// TwinCAT 3 PLC project P_Connect
// ProgramVersion: 3.1.4023.0
// libraries:
//   Tc2_EIB, * (Beckhoff Automation GmbH)
//   Tc2_IoFunctions, * (Beckhoff Automation GmbH)
//   Tc2_MBus, * (Beckhoff Automation GmbH)
//   Tc2_SerialCom, * (Beckhoff Automation GmbH)
//   Tc2_Standard, * (Beckhoff Automation GmbH)
//   Tc2_System, * (Beckhoff Automation GmbH)
//   Tc3_Module, * (Beckhoff Automation GmbH)
// project tree:
//   DUTs/ st_P_Connect_to_Lynus.TcDUT
//   GVLs/ Global_var.TcGVL, GVL_EfficientIO.TcGVL, p_Datenschnittstelle.TcPOU
//   / PlcTask.TcTTO
//   POUs/ MAIN.TcPOU
// real-time tasks:
//   TASK PlcTask: cycle T#10ms, priority 20, ADS port 350
//   TASK EfficientIO_Communication: cycle T#5ms, priority 15, ADS port 351
//   TASK PlcTask1: cycle T#10ms, priority 21, ADS port 353
// variable links:
//   Lynus_Test/Lynus_Test Instance <-> P_Connect/P_Connect Instance
//     PlcTask1 Inputs/GVL.lynus_in <-> PlcTask Outputs/GVL_EfficientIO.lynus_out
//     PlcTask1 Outputs/GVL.lynus_out <-> PlcTask Inputs/GVL_EfficientIO.lynus_in

CONFIGURATION P_Connect
    RESOURCE PLC ON TwinCAT3
        TASK PlcTask(INTERVAL := T#10ms, PRIORITY := 20);
        PROGRAM MAIN WITH PlcTask : MAIN;
    END_RESOURCE
END_CONFIGURATION

// ---- DUTs/st_P_Connect_to_Lynus.TcDUT
TYPE st_P_Connect_to_Lynus :
STRUCT
	Wert_1	:REAL;	
	Wert_2	:REAL;	
	Wert_3	:REAL;	
	Wert_4	:REAL;	
	Wert_5	:REAL;	
	Wert_6	:REAL;	
	Wert_7	:BOOL;	
	Wert_8	:REAL;	
	Wert_9	:REAL;	
	Wert_10	:REAL;
	Wert_11	:REAL;	
	Wert_12	:REAL;	
	Wert_13	:REAL;	
	Wert_14	:REAL;	
	Wert_15	:REAL;	
	Wert_16	:REAL;	
	Wert_17	:REAL;	
	Wert_18	:REAL;	
	Wert_19	:REAL;	
	Wert_20	:REAL;
	Wert_21	:REAL;	
	Wert_22	:REAL;	
	Wert_23	:REAL;	
	Wert_24	:REAL;	
	Wert_25	:REAL;	
	Wert_26	:REAL;	
	Wert_27	:REAL;	
	Wert_28	:REAL;	
	Wert_29	:REAL;	
	Wert_30	:REAL;
	Wert_31	:REAL;
	Wert_32	:REAL;
	Wert_33	:REAL;
	Wert_34	:REAL;
	Wert_35	:REAL;
	Wert_36	:REAL;
	Wert_37	:REAL;
	Wert_38	:REAL;
	Wert_39	:REAL;
	Wert_40	:REAL;
	Wert_41	:BOOL;
	Wert_42	:BOOL;
	Wert_43	:BOOL;
	Wert_44	:BOOL;
	Wert_45	:BOOL;
	Wert_46	:BOOL;
	Wert_47	:BOOL;
	Wert_48	:BOOL;
	Wert_49	:BOOL;
	Wert_50	:BOOL;
	Wert_51	:BOOL;
	Wert_52	:BOOL;
END_STRUCT
END_TYPE

// ---- GVLs/Global_var.TcGVL
VAR_GLOBAL
	_ARRAY_IP			:ARRAY [1..50] OF STRING; 
	_ARRAY_name_of_var	:ARRAY [1..50] OF STRING(255);
	_ARRAY_var_value	:ARRAY [1..50] OF REAL;
END_VAR

// ---- GVLs/GVL_EfficientIO.TcGVL
{attribute 'qualified_only'}
VAR_GLOBAL
	lynus_out   				AT %Q* 	: st_P_Connect_to_Lynus;
	lynus_in   					AT %I* 	: st_P_Connect_to_Lynus;	
	
	(*KNX*)
	TEMP_INNEN_1			:REAL;	
	RH_INNEN_1				:REAL;	
	TEMP_INNEN_2			:REAL;	
	RH_INNEN_2				:REAL;	
	TEMP_AUSSEN				:REAL;	
	RH_AUSSEN				:REAL;		
	AKTIVITAET				:BOOL;
	
	(*M-Bus variablen für Lynus*)
	ELEKTRO_1_Zaehler		:REAL;
	ELEKTRO_1_Leistung		:REAL;
	ELEKTRO_2_Zaehler		:REAL;
	ELEKTRO_2_Leistung		:REAL;
	ELEKTRO_3_Zaehler		:REAL;
	ELEKTRO_3_Leistung		:REAL;
	ELEKTRO_4_Zaehler		:REAL;
	ELEKTRO_4_Leistung		:REAL;
	ELEKTRO_5_Zaehler		:REAL;
	ELEKTRO_5_Leistung		:REAL;
	HEIZEN					:REAL;
	
	(*IMPULSZÄHLER*)
	Wasseruhr_1				:REAL;
	Wasseruhr_2				:REAL;

	(*PT1000 Temp.*)
	TEMP_HKLS_1				:REAL;
	TEMP_HKLS_2				:REAL;
	TEMP_HKLS_3				:REAL;
	TEMP_HKLS_4				:REAL;
	TEMP_HKLS_5				:REAL; 
	TEMP_HKLS_6				:REAL;
	TEMP_HKLS_7				:REAL;
	TEMP_HKLS_8				:REAL;
	
	(*Zentalfunktionen*)
	VERSCHATTUNG_auf		:BOOL;
	VERSCHATTUNG_ab			:BOOL;
	ZENTRAL_LICHT_ein_EG	:BOOL;
	ZENTRAL_LICHT_aus_EG	:BOOL;
	ZENTRAL_LICHT_ein_OG	:BOOL;
	ZENTRAL_LICHT_aus_OG	:BOOL;
	BA3_ZENTRAL_LICHT_ein	:BOOL;
	BA3_ZENTRAL_LICHT_aus	:BOOL;
	BA3_VERSCHATTUNG_auf_EG	:BOOL;
	BA3_VERSCHATTUNG_ab_EG	:BOOL;
	BA3_VERSCHATTUNG_auf_OG	:BOOL;
	BA3_VERSCHATTUNG_ab_OG	:BOOL;
END_VAR

// ---- POUs/MAIN.TcPOU
PROGRAM MAIN
VAR

l_ton_Trigger_Auslesen			: TON;
l_ton_Trigger_Auslesen_BOOL		: TON;

l_tp_VERSCHATTUNG_auf		: TP;
l_tp_VERSCHATTUNG_ab		: TP;
l_tp_ZENTRAL_LICHT_ein_EG	: TP;
l_tp_ZENTRAL_LICHT_aus_EG	: TP;
l_tp_ZENTRAL_LICHT_ein_OG	: TP;
l_tp_ZENTRAL_LICHT_aus_OG	: TP;

l_BA3_tp_VERSCHATTUNG_auf_OG	: TP;
l_BA3_tp_VERSCHATTUNG_ab_OG		: TP;
l_BA3_tp_VERSCHATTUNG_auf_EG	: TP;
l_BA3_tp_VERSCHATTUNG_ab_EG		: TP;
l_BA3_tp_ZENTRAL_LICHT_ein		: TP;
l_BA3_tp_ZENTRAL_LICHT_aus		: TP;



l_fb_ADS_read_HK_LA 		: ADSRDWRTEX; 
l_fb_ADS_read_HK_LA_BOOL	: ADSRDWRTEX; 

i :INT:= 1;
l_b_only_once	:BOOL;
l_b_test		:BOOL;
l_r_destaddr	:REAL;
gv_PCon_bAktivitaet_EG_OG :BOOL;
END_VAR

_ARRAY_IP[1] := '10.0.0.10.1.1';
_ARRAY_name_of_var[1] := '.p_machineParameter_i1.ToZpoint.ProductDataAttributes_EZ_Gesamtzaehler_i1.EZ_Gesamtzaehler_Zaehlerwerte_1_ov_r_Wirkenergie_positivTotal.r_value';

_ARRAY_IP[2] := '10.0.0.10.1.1';
_ARRAY_name_of_var[2] := '.p_machineParameter_i1.ToZpoint.ProductDataAttributes_EZ_Gesamtzaehler_i1.EZ_Gesamtzaehler_Zaehlerwerte_1_ov_r_Wirkleistung_positivTotal.r_value';

_ARRAY_IP[3] := '10.0.0.10.1.1';
_ARRAY_name_of_var[3] := '.p_machineParameter_i1.ToZpoint.ProductDataAttributes_EZ_Waermepumpe_1_i1.EZ_Waermepumpe_1_Zaehlerwerte_ov_r_EnergyTotal.r_value';

_ARRAY_IP[4] := '10.0.0.10.1.1';
_ARRAY_name_of_var[4] := '.p_machineParameter_i1.ToZpoint.ProductDataAttributes_EZ_Waermepumpe_1_i1.EZ_Waermepumpe_1_Zaehlerwerte_ov_r_Wirkleistung.r_value';

_ARRAY_IP[5] := '10.0.0.10.1.1';
_ARRAY_name_of_var[5] := '.p_machineParameter_i1.ToZpoint.ProductDataAttributes_EZ_Waermepumpe_2_i1.EZ_Waermepumpe_2_Zaehlerwerte_ov_r_EnergyTotal.r_value';

_ARRAY_IP[6] := '10.0.0.10.1.1';
_ARRAY_name_of_var[6] := '.p_machineParameter_i1.ToZpoint.ProductDataAttributes_EZ_Waermepumpe_2_i1.EZ_Waermepumpe_2_Zaehlerwerte_ov_r_Wirkleistung.r_value';

_ARRAY_IP[7] := '10.0.0.10.1.1';
_ARRAY_name_of_var[7] := '.p_machineParameter_i1.ToZpoint.ProductDataAttributes_EZ_Ladestation_1_i1.EZ_Ladestation_1_Zaehlerwerte_ov_r_EnergyTotal.r_value';

_ARRAY_IP[8] := '10.0.0.10.1.1';
_ARRAY_name_of_var[8] := '.p_machineParameter_i1.ToZpoint.ProductDataAttributes_EZ_Ladestation_1_i1.EZ_Ladestation_1_Zaehlerwerte_ov_r_Wirkleistung.r_value';

_ARRAY_IP[9] := '10.0.0.10.1.1';
_ARRAY_name_of_var[9] := '.p_machineParameter_i1.ToZpoint.ProductDataAttributes_EZ_Ladestation_2_i1.EZ_Ladestation_2_Zaehlerwerte_ov_r_EnergyTotal.r_value';

_ARRAY_IP[10] := '10.0.0.10.1.1';
_ARRAY_name_of_var[10] := '.p_machineParameter_i1.ToZpoint.ProductDataAttributes_EZ_Ladestation_2_i1.EZ_Ladestation_2_Zaehlerwerte_ov_r_Wirkleistung.r_value';

_ARRAY_IP[11] := '10.0.0.10.1.1';
_ARRAY_name_of_var[11] := '.p_machineParameter_i1.ToZpoint.ProductDataAttributes_EZ_Ladestation_5_i1.EZ_Ladestation_5_Zaehlerwerte_ov_r_EnergyTotal.r_value';

_ARRAY_IP[12] := '10.0.0.10.1.1';
_ARRAY_name_of_var[12] := '.p_machineParameter_i1.ToZpoint.ProductDataAttributes_EZ_Ladestation_5_i1.EZ_Ladestation_5_Zaehlerwerte_ov_r_Wirkleistung.r_value';

_ARRAY_IP[13] := '10.0.0.10.1.1';
_ARRAY_name_of_var[13] := '.p_machineParameter_i1.ToZpoint.ProductDataAttributes_EZ_PV_Anlage_i1.EZ_PV_Wechselrichter_1_ov_r_ErzeugteWirkenergie.r_value';

_ARRAY_IP[14] := '10.0.0.10.1.1';
_ARRAY_name_of_var[14] := '.p_machineParameter_i1.ToZpoint.ProductDataAttributes_EZ_PV_Anlage_i1.EZ_PV_Wechselrichter_1_ov_r_Wirkleistung.r_value';

_ARRAY_IP[15] := '10.0.0.10.1.1';
_ARRAY_name_of_var[15] := '.p_machineParameter_i1.ToZpoint.ProductDataAttributes_EZ_PV_Anlage_i1.EZ_PV_Wechselrichter_2_ov_r_ErzeugteWirkenergie.r_value';

_ARRAY_IP[16] := '10.0.0.10.1.1';
_ARRAY_name_of_var[16] := '.p_machineParameter_i1.ToZpoint.ProductDataAttributes_EZ_PV_Anlage_i1.EZ_PV_Wechselrichter_2_ov_r_Wirkleistung.r_value';

_ARRAY_IP[17] := '10.0.0.10.1.1';
_ARRAY_name_of_var[17] := '.p_machineParameter_i1.ToZpoint.ProductDataAttributes_WMZ_01_Gaskessel_i1.WMZ_01_Gaskessel_Normaltarif_ov_r_EnergyTarif.r_value';

_ARRAY_IP[18] := '10.0.0.10.1.1';
_ARRAY_name_of_var[18] := '.p_machineParameter_i1.ToZpoint.ProductDataAttributes_WMZ_01_Gaskessel_i1.WMZ_01_Gaskessel_ov_r_Power.r_value';

_ARRAY_IP[19] := '10.0.0.10.1.1';
_ARRAY_name_of_var[19] := '.p_machineParameter_i1.ToZpoint.ProductDataAttributes_WMZ_03_WT01_WP_i1.WMZ_03_Waermetauscher_1_WP_ov_r_Power.r_value';

_ARRAY_IP[20] := '10.0.0.10.1.1';
_ARRAY_name_of_var[20] := '.p_machineParameter_i1.ToZpoint.ProductDataAttributes_WMZ_03_WT01_WP_i1.WMZ_03_Waermetauscher_1_WP_Normaltarif_ov_r_EnergyTarif.r_value';

_ARRAY_IP[21] := '10.0.0.10.1.1';
_ARRAY_name_of_var[21] := '.p_machineParameter_i1.ToZpoint.ProductDataAttributes_WMZ_03_WT01_WP_i1.WMZ_03_Waermetauscher_1_WP_Tarif_1_ov_r_EnergyTarif.r_value';

//notdonecontrolle
_ARRAY_IP[22] := '10.0.0.20.1.1';
_ARRAY_name_of_var[22] := '.p_machineParameter_i1.ToZpoint.Visualisierung_Wettersation_i1.Wettersation.Wetterstation_1.Temperatur.ov_r_Data';

_ARRAY_IP[23] := '10.0.0.20.1.1';
_ARRAY_name_of_var[23] := '.p_machineParameter_i1.ToZpoint.ProductDataAttributes_LA_Temperatursensoren_i1.LA_Temperatursensoren_Temperatur_Zuluft_ov_r_valueCorrected.r_value';

_ARRAY_IP[24] := '10.0.0.20.1.1';
_ARRAY_name_of_var[24] := '.p_machineParameter_i1.ToZpoint.ProductDataAttributes_Raum_104_Buero_2_i1.Raum_104_Buero_2_ov_rRaumtemperatur.r_value';

_ARRAY_IP[25] := '10.0.0.20.1.1';
_ARRAY_name_of_var[25] := '.p_machineParameter_i1.ToZpoint.ProductDataAttributes_Halle_027_Montage_i1.Halle_027_Montage_ov_rRaumtemperatur.r_value';

_ARRAY_IP[26] := '10.0.0.20.1.1';
_ARRAY_name_of_var[26] := '.p_machineParameter_i1.ToZpoint.ProductDataAttributes_Raum_025_Mehrzweck_und_Aufenthaltsraum_i1.Raum_025_Mehrzweck_und_Aufenthaltsraum_ov_rRaumtemperatur.r_value';

_ARRAY_IP[27] := '10.0.0.10.1.1';
_ARRAY_name_of_var[27] := '.p_machineParameter_i1.ToZpoint.ProductDataAttributes_EZ_Gesamtzaehler_i1.EZ_Gesamtzaehler_Zaehlerwerte_1_ov_r_Wirkenergie_nagativTotal.r_value';

_ARRAY_IP[28] := '10.0.0.10.1.1';
_ARRAY_name_of_var[28] := '.p_machineParameter_i1.ToZpoint.ProductDataAttributes_EZ_Gesamtzaehler_i1.EZ_Gesamtzaehler_Zaehlerwerte_1_ov_r_Wirkleistung_nagativTotal.r_value';

_ARRAY_IP[29] := '10.0.0.10.1.1';
_ARRAY_name_of_var[29] := '.p_machineParameter_i1.ToZpoint.ProductDataAttributes_EZ_PV_Anlage_i1.EZ_PV_Wechselrichter_3_ov_r_ErzeugteWirkenergie.r_value';

_ARRAY_IP[30] := '10.0.0.10.1.1';
_ARRAY_name_of_var[30] := '.p_machineParameter_i1.ToZpoint.ProductDataAttributes_EZ_PV_Anlage_i1.EZ_PV_Wechselrichter_3_ov_r_Wirkleistung.r_value';

_ARRAY_IP[31] := '10.0.0.10.1.1';
_ARRAY_name_of_var[31] := '.p_machineParameter_i1.ToZpoint.ProductDataAttributes_EZ_PV_Anlage_i1.EZ_PV_Wechselrichter_4_ov_r_ErzeugteWirkenergie.r_value';

_ARRAY_IP[32] := '10.0.0.10.1.1';
_ARRAY_name_of_var[32] := '.p_machineParameter_i1.ToZpoint.ProductDataAttributes_EZ_PV_Anlage_i1.EZ_PV_Wechselrichter_4_ov_r_Wirkleistung.r_value';

_ARRAY_IP[33] := '10.0.0.10.1.1';
_ARRAY_name_of_var[33] := '.p_machineParameter_i1.ToZpoint.ProductDataAttributes_EZ_PV_Anlage_i1.EZ_PV_Wechselrichter_5_ov_r_ErzeugteWirkenergie.r_value';

_ARRAY_IP[34] := '10.0.0.10.1.1';
_ARRAY_name_of_var[34] := '.p_machineParameter_i1.ToZpoint.ProductDataAttributes_EZ_PV_Anlage_i1.EZ_PV_Wechselrichter_5_ov_r_Wirkleistung.r_value';

_ARRAY_IP[35] := '10.0.0.10.1.1';
_ARRAY_name_of_var[35] := '.p_machineParameter_i1.ToZpoint.ProductDataAttributes_EZ_PV_Anlage_i1.EZ_PV_Wechselrichter_6_ov_r_ErzeugteWirkenergie.r_value';

_ARRAY_IP[36] := '10.0.0.10.1.1';
_ARRAY_name_of_var[36] := '.p_machineParameter_i1.ToZpoint.ProductDataAttributes_EZ_PV_Anlage_i1.EZ_PV_Wechselrichter_6_ov_r_Wirkleistung.r_value';

_ARRAY_IP[37] := '10.0.0.10.1.1';
_ARRAY_name_of_var[37] := '.p_machineParameter_i1.ToZpoint.ProductDataAttributes_EZ_PV_Anlage_i1.EZ_PV_Wechselrichter_7_ov_r_ErzeugteWirkenergie.r_value';

_ARRAY_IP[38] := '10.0.0.10.1.1';
_ARRAY_name_of_var[38] := '.p_machineParameter_i1.ToZpoint.ProductDataAttributes_EZ_PV_Anlage_i1.EZ_PV_Wechselrichter_7_ov_r_Wirkleistung.r_value';

_ARRAY_IP[39] := '10.0.0.10.1.1';
_ARRAY_name_of_var[39] := '.p_machineParameter_i1.ToZpoint.ProductDataAttributes_EZ_PV_Anlage_i1.EZ_PV_Wechselrichter_8_ov_r_ErzeugteWirkenergie.r_value';

_ARRAY_IP[40] := '10.0.0.10.1.1';
_ARRAY_name_of_var[40] := '.p_machineParameter_i1.ToZpoint.ProductDataAttributes_EZ_PV_Anlage_i1.EZ_PV_Wechselrichter_8_ov_r_Wirkleistung.r_value';

_ARRAY_IP[41] := '10.0.0.10.1.1';
_ARRAY_name_of_var[41] := '.p_machineParameter_i1.ToZpoint.ProductDataAttributes_EZ_PV_Anlage_i1.EZ_PV_Wechselrichter_9_ov_r_ErzeugteWirkenergie.r_value';

_ARRAY_IP[42] := '10.0.0.10.1.1';
_ARRAY_name_of_var[42] := '.p_machineParameter_i1.ToZpoint.ProductDataAttributes_EZ_PV_Anlage_i1.EZ_PV_Wechselrichter_9_ov_r_Wirkleistung.r_value';

//BA3 WP aktulle leistung
_ARRAY_IP[43] := '10.0.0.30.1.1';
_ARRAY_name_of_var[43] := '.p_machineParameter_i1.ToZpoint.ProductDataAttributes_WMZ02_Waermepumpe_BA3E_i1.WMZ02_Waermepumpe_BA3E_ov_r_Power.r_value'; 
//BA3 WP Wärme Energie
_ARRAY_IP[44] := '10.0.0.30.1.1';
_ARRAY_name_of_var[44] := '.p_machineParameter_i1.ToZpoint.ProductDataAttributes_WMZ02_Waermepumpe_BA3E_i1.WMZ02_Waermepumpe_BA3E_ov_r_EnergyT1.r_value';
//BA3 Kälte Energie
_ARRAY_IP[45] := '10.0.0.30.1.1';
_ARRAY_name_of_var[45] := '.p_machineParameter_i1.ToZpoint.ProductDataAttributes_WMZ02_Waermepumpe_BA3E_i1.WMZ02_Waermepumpe_BA3E_ov_r_EnergyT2.r_value';

//BA3 Wasserzähler
_ARRAY_IP[46] := '10.0.0.10.1.1';
_ARRAY_name_of_var[46] := '.p_machineParameter_i1.ToZpoint.ProductDataAttributes_WZ_Wasserzaehler_Gesamt_i1.WZ_Wasserzaehler_Gesamt_ov_r_Volume.r_value';
//BA3 Wasserzähler
_ARRAY_IP[47] := '10.0.0.10.1.1';
_ARRAY_name_of_var[47] := '.p_machineParameter_i1.ToZpoint.ProductDataAttributes_WZ_Wasserzaehler_Gesamt_i1.WZ_Wasserzaehler_Gesamt_ov_r_Flow.r_value';

l_ton_Trigger_Auslesen	(PT:= T#400MS);

//KNX Signale senden/ via ADS and Bestands GLT
l_tp_VERSCHATTUNG_auf	(PT:= T#2000MS,
						 IN:=GVL_EfficientIO.lynus_in.Wert_41, 
						 Q=>GVL_EfficientIO.VERSCHATTUNG_auf);
						 
l_tp_VERSCHATTUNG_ab	(PT:= T#2000MS,
						 IN:=GVL_EfficientIO.lynus_in.Wert_42,
						 Q=> GVL_EfficientIO.VERSCHATTUNG_ab);
						 
l_tp_ZENTRAL_LICHT_ein_EG	(PT:= T#2000MS,
							 IN:= GVL_EfficientIO.lynus_in.Wert_43, 
							 Q=>  GVL_EfficientIO.ZENTRAL_LICHT_ein_EG);
						 
l_tp_ZENTRAL_LICHT_aus_EG	(PT:= T#2000MS,
							 IN:= GVL_EfficientIO.lynus_in.Wert_44, 
							 Q=>  GVL_EfficientIO.ZENTRAL_LICHT_aus_EG);
							 
l_tp_ZENTRAL_LICHT_ein_OG	(PT:= T#2000MS,
							 IN:= GVL_EfficientIO.lynus_in.Wert_45, 
							 Q=>  GVL_EfficientIO.ZENTRAL_LICHT_ein_OG);
						 
l_tp_ZENTRAL_LICHT_aus_OG	(PT:= T#2000MS,
							 IN:= GVL_EfficientIO.lynus_in.Wert_46, 
							 Q=>  GVL_EfficientIO.ZENTRAL_LICHT_aus_OG);
							 
//BA3							 
l_BA3_tp_VERSCHATTUNG_ab_OG(PT:= T#2000MS,
							 IN:= GVL_EfficientIO.lynus_in.Wert_51, 
							 Q=>  GVL_EfficientIO.BA3_VERSCHATTUNG_ab_OG);
							 
l_BA3_tp_VERSCHATTUNG_auf_OG(PT:= T#2000MS,
							 IN:= GVL_EfficientIO.lynus_in.Wert_52, 
							 Q=>  GVL_EfficientIO.BA3_VERSCHATTUNG_auf_OG);
							 
l_BA3_tp_VERSCHATTUNG_auf_EG(PT:= T#2000MS,
							 IN:= GVL_EfficientIO.lynus_in.Wert_50, 
							 Q=>  GVL_EfficientIO.BA3_VERSCHATTUNG_auf_EG);

l_BA3_tp_VERSCHATTUNG_ab_EG(PT:= T#2000MS,
							 IN:= GVL_EfficientIO.lynus_in.Wert_49, 
							 Q=>  GVL_EfficientIO.BA3_VERSCHATTUNG_ab_EG);

l_BA3_tp_ZENTRAL_LICHT_ein(PT:= T#2000MS,
							 IN:= GVL_EfficientIO.lynus_in.Wert_47, 
							 Q=>  GVL_EfficientIO.BA3_ZENTRAL_LICHT_ein);

l_BA3_tp_ZENTRAL_LICHT_aus(PT:= T#2000MS,
							 IN:= GVL_EfficientIO.lynus_in.Wert_48, 
							 Q=>  GVL_EfficientIO.BA3_ZENTRAL_LICHT_aus);					 
							 
IF NOT l_fb_ADS_read_HK_LA.BUSY AND l_ton_Trigger_Auslesen.Q THEN
	IF  i = 47 THEN
		i := 1;
	ELSE	
		i := i+1;
	END_IF
	l_ton_Trigger_Auslesen.IN:= FALSE;
ELSE
	l_ton_Trigger_Auslesen.IN:= TRUE;
END_IF
	
l_fb_ADS_read_HK_LA(
NETID:=		_ARRAY_IP[i],
PORT:= 		801, 
IDXGRP:= 	16#F004, 
IDXOFFS:= 	0, 
WRITELEN:=	LEN(_ARRAY_name_of_var[i]),
READLEN :=	SIZEOF(REAL),
SRCADDR:= 	ADR(_ARRAY_name_of_var[i]), 
DESTADDR:=	ADR(_ARRAY_var_value[i]),
WRTRD:= 	NOT l_ton_Trigger_Auslesen.Q, 
TMOUT:= 	T#1S
);

l_ton_Trigger_Auslesen_BOOL	(PT:= T#3000MS);

IF NOT l_fb_ADS_read_HK_LA_BOOL.BUSY AND l_ton_Trigger_Auslesen_BOOL.Q THEN
	l_ton_Trigger_Auslesen_BOOL.IN:= FALSE;
ELSE
	l_ton_Trigger_Auslesen_BOOL.IN:= TRUE;
END_IF

l_fb_ADS_read_HK_LA_BOOL(
NETID:=		'10.0.0.20.1.1',
PORT:= 		801, 
IDXGRP:= 	16#F004, 
IDXOFFS:= 	0, 
WRITELEN:=	LEN('.gv_PCon_bAktivitaet_EG_OG'),
READLEN :=	SIZEOF(BOOL),
SRCADDR:= 	ADR('.gv_PCon_bAktivitaet_EG_OG'), 
DESTADDR:=	ADR(GVL_EfficientIO.AKTIVITAET),
WRTRD:= 	NOT l_ton_Trigger_Auslesen_BOOL.Q, 
TMOUT:= 	T#3S
);	

p_Datenschnittstelle();

END_PROGRAM

// ---- GVLs/p_Datenschnittstelle.TcPOU
PROGRAM p_Datenschnittstelle
VAR
	l_r_summe_WP1_WP2_kWH			:REAL;
	l_r_summe_WP1_WP2_kW			:REAL;
	l_r_summe_Ladestation_1_2_5_kWh	:REAL;
	l_r_summe_Ladestation_1_2_5_kW	:REAL;
	l_r_summe_PV1_PV2_kWh			:REAL;
	l_r_summe_PV1_PV2_kW			:REAL;
	l_r_summe_gessamt_Pos_und_gesamt_neg_kW :REAL;
	Test_2_1 : REAL;
	Test_2_2 : REAL;
	Test_2_3 : REAL;
END_VAR

//GVL_EfficientIO.lynusinout.Wert_1	:=;
//GVL_EfficientIO.lynusinout.Wert_2	:=;
//GVL_EfficientIO.lynusinout.Wert_3	:=;
//GVL_EfficientIO.lynusinout.Wert_4	:=;
//GVL_EfficientIO.lynusinout.Wert_5	:=;
GVL_EfficientIO.lynus_out.Wert_6	:=_ARRAY_var_value[27];
GVL_EfficientIO.lynus_out.Wert_7	:=GVL_EfficientIO.AKTIVITAET;
GVL_EfficientIO.lynus_out.Wert_8	:=_ARRAY_var_value[1];
GVL_EfficientIO.lynus_out.Wert_9	:=l_r_summe_gessamt_Pos_und_gesamt_neg_kW;
GVL_EfficientIO.lynus_out.Wert_10	:=l_r_summe_WP1_WP2_kWH;
GVL_EfficientIO.lynus_out.Wert_11	:=l_r_summe_WP1_WP2_kW;
GVL_EfficientIO.lynus_out.Wert_12	:=l_r_summe_Ladestation_1_2_5_kWh;
GVL_EfficientIO.lynus_out.Wert_13	:=l_r_summe_Ladestation_1_2_5_kW;
GVL_EfficientIO.lynus_out.Wert_14	:=l_r_summe_PV1_PV2_kWh;
GVL_EfficientIO.lynus_out.Wert_15	:=l_r_summe_PV1_PV2_kW;
GVL_EfficientIO.lynus_out.Wert_16	:=_ARRAY_var_value[17];
GVL_EfficientIO.lynus_out.Wert_17	:=_ARRAY_var_value[18];
//GVL_EfficientIO.lynus_out.Wert_18	:=_ARRAY_var_value[43];
//GVL_EfficientIO.lynus_out.Wert_19	:=_ARRAY_var_value[44];
GVL_EfficientIO.lynus_out.Wert_20	:=_ARRAY_var_value[46];
GVL_EfficientIO.lynus_out.Wert_21	:=_ARRAY_var_value[47];
GVL_EfficientIO.lynus_out.Wert_22	:=_ARRAY_var_value[22];
GVL_EfficientIO.lynus_out.Wert_23	:=_ARRAY_var_value[23];
GVL_EfficientIO.lynus_out.Wert_24	:=_ARRAY_var_value[24];
GVL_EfficientIO.lynus_out.Wert_25	:=_ARRAY_var_value[25];
GVL_EfficientIO.lynus_out.Wert_26	:=_ARRAY_var_value[26];
GVL_EfficientIO.lynus_out.Wert_27	:=_ARRAY_var_value[19];
GVL_EfficientIO.lynus_out.Wert_28	:=_ARRAY_var_value[20];
GVL_EfficientIO.lynus_out.Wert_29	:=_ARRAY_var_value[21];
GVL_EfficientIO.lynus_out.Wert_30	:=_ARRAY_var_value[8];
GVL_EfficientIO.lynus_out.Wert_31	:=_ARRAY_var_value[43];
GVL_EfficientIO.lynus_out.Wert_32	:=_ARRAY_var_value[44];
GVL_EfficientIO.lynus_out.Wert_33	:=_ARRAY_var_value[45];

l_r_summe_WP1_WP2_kWH 			:= _ARRAY_var_value[3] + _ARRAY_var_value[5]; 
l_r_summe_WP1_WP2_kW 			:= (_ARRAY_var_value[4]) + (_ARRAY_var_value[6]);
l_r_summe_Ladestation_1_2_5_kWh	:= (_ARRAY_var_value[7]) + (_ARRAY_var_value[9]) + (_ARRAY_var_value[11]);
l_r_summe_Ladestation_1_2_5_kW	:= (_ARRAY_var_value[8]) + (_ARRAY_var_value[10]) +(_ARRAY_var_value[12]);
l_r_summe_PV1_PV2_kWh			:= (_ARRAY_var_value[13]) + (_ARRAY_var_value[15]) + (_ARRAY_var_value[29]) + (_ARRAY_var_value[31]) + (_ARRAY_var_value[33]) + (_ARRAY_var_value[35]) + (_ARRAY_var_value[37]) + (_ARRAY_var_value[39]) + (_ARRAY_var_value[41]);
l_r_summe_PV1_PV2_kW			:= (_ARRAY_var_value[14]) + (_ARRAY_var_value[16]) + (_ARRAY_var_value[30]) + (_ARRAY_var_value[32]) + (_ARRAY_var_value[34]) + (_ARRAY_var_value[36]) + (_ARRAY_var_value[38]) + (_ARRAY_var_value[40]) + (_ARRAY_var_value[42]);
l_r_summe_gessamt_Pos_und_gesamt_neg_kW :=(_ARRAY_var_value[2]) - (_ARRAY_var_value[28]);

GVL_EfficientIO.VERSCHATTUNG_auf		:=GVL_EfficientIO.lynus_in.Wert_41;
GVL_EfficientIO.VERSCHATTUNG_ab			:=GVL_EfficientIO.lynus_in.Wert_42;
GVL_EfficientIO.ZENTRAL_LICHT_ein_EG	:=GVL_EfficientIO.lynus_in.Wert_43;
GVL_EfficientIO.ZENTRAL_LICHT_aus_EG	:=GVL_EfficientIO.lynus_in.Wert_44;
GVL_EfficientIO.ZENTRAL_LICHT_ein_OG	:=GVL_EfficientIO.lynus_in.Wert_45;
GVL_EfficientIO.ZENTRAL_LICHT_aus_OG	:=GVL_EfficientIO.lynus_in.Wert_46;
(*
GVL_EfficientIO.BA3_ZENTRAL_LICHT_ein 	:=GVL_EfficientIO.lynus_in.Wert_47;
GVL_EfficientIO.BA3_ZENTRAL_LICHT_aus	:=GVL_EfficientIO.lynus_in.Wert_48;
GVL_EfficientIO.BA3_VERSCHATTUNG_auf_EG :=GVL_EfficientIO.lynus_in.Wert_49;
GVL_EfficientIO.BA3_VERSCHATTUNG_ab_EG 	:=GVL_EfficientIO.lynus_in.Wert_50;
GVL_EfficientIO.BA3_VERSCHATTUNG_auf_OG	:=GVL_EfficientIO.lynus_in.Wert_51;
GVL_EfficientIO.BA3_VERSCHATTUNG_ab_OG	:=GVL_EfficientIO.lynus_in.Wert_52;*)

END_PROGRAM
